TYPE ST_BigBagChangeHandlerInCmd :
STRUCT
    bConfirmBagChange   : BOOL;   // potwierdzenie operatora, że nowy worek został założony
END_STRUCT
END_TYPE

(* stored: Version 1.1.0.1, ProductVersion 3.1.4024.16
   DUT ST_BigBagChangeHandlerInCmd: Id {cf7b336d-c889-4935-8263-3d19db32019c} *)
